{attribute 'linkalways'} 
{attribute 'no_explicit_call' := 'This FB is a CLASS and must be accessed using methods or properties'}
{attribute 'enable_dynamic_creation'}
FUNCTION_BLOCK Node_F_VN_DistanceTransformationExp EXTENDS VisionNode
VAR
    ipSrcImage : _ITcVnImage;
    ipDestImage : _ITcVnImage;
    eDistanceType : _ETcVnDistanceType(ETcVnDistanceType.TCVN_DT_L1);
    eMaskSize : _ETcVnDistanceTransformationMask(ETcVnDistanceTransformationMask.TCVN_DTM_PRECISE);
    ipDestLabels : _ITcVnImage;
    eLabelType : _ETcVnDistanceTransformationLabel(ETcVnDistanceTransformationLabel.TCVN_DTL_CCOMP);
    hrPrev : _HRESULT(S_OK);
	hresult : _HRESULT(S_OK);
END_VAR

METHOD PUBLIC  Clone : I_Node
VAR
	pNode : POINTER TO Node_F_VN_DistanceTransformationExp;
END_VAR
pNode := __NEW(Node_F_VN_DistanceTransformationExp);
Clone := pNode^;
END_METHOD

METHOD FB_init : BOOL
VAR_INPUT
	bInitRetains : BOOL; // if TRUE, the retain variables are initialized (warm start / cold start)
	bInCopyCode : BOOL;  // if TRUE, the instance afterwards gets moved into the copy code (online change)
END_VAR
AddInput('ipSrcImage', ipSrcImage);
AddParameter('eDistanceType', eDistanceType);
AddParameter('eMaskSize', eMaskSize);
AddParameter('eLabelType', eLabelType);
AddInput('hrPrev', hrPrev);
AddOutput('ipDestImage', ipDestImage);
AddOutput('ipDestLabels', ipDestLabels);
AddOutput('hresult',hresult);
END_METHOD

METHOD PROTECTED OnExecute
hresult.Value := F_VN_DistanceTransformationExp(
    ipSrcImage := ipSrcImage.Value,
	ipDestImage := ipDestImage.Value,
    eDistanceType := eDistanceType.Value,
    eMaskSize := eMaskSize.Value,
    ipDestLabels := ipDestLabels.Value,
    eLabelType := eLabelType.Value,
	hrPrev:= hrPrev.Value);
END_METHOD

METHOD PUBLIC PreExecutionCheck
VAR_INPUT
	Check : I_PreExecutionChecks;
END_VAR
VAR
    distanceTypeIsValid : BOOL;
    maskSizeIsValid : BOOL;
END_VAR
Check.IsTrue(ipSrcImage.IsValid, 'ipSrcImage must contain an image');
Check.IsTrue(ipSrcImage.HasChannelCount(1), 'ipSrcImage must have 1 channel');
Check.IsTrue(ipSrcImage.IsPixelDepth(8), 'ipSrcImage must have 8 bit pixel depth');

CASE eDistanceType.Value OF
    ETcVnDistanceType.TCVN_DT_L1,
    ETcVnDistanceType.TCVN_DT_L2,
    ETcVnDistanceType.TCVN_DT_C :
        distanceTypeIsValid := TRUE;
END_CASE
Check.IsTrue(distanceTypeIsValid, 'eDistanceType value is unsupported');

CASE eMaskSize.Value OF
    ETcVnDistanceTransformationMask.TCVN_DTM_3,
    ETcVnDistanceTransformationMask.TCVN_DTM_5 :
        maskSizeIsValid := TRUE;
END_CASE
Check.IsTrue(maskSizeIsValid, 'maskSizeIsValid value is unsupported');
END_METHOD

END_FUNCTION_BLOCK

(* stored: Version 1.1.0.1, ProductVersion 3.1.4024.15
   POU Node_F_VN_DistanceTransformationExp: Id {ff2c9989-7375-4244-a20d-67b814b76b41}, SpecialFunc None
   Folder Constructor: Id {0ac6e05f-fa8b-473e-b8a7-f4d93839d812}
   Method Clone: Id {a38c76e1-8bd5-471a-9be6-96e8afdf7058}
   Method FB_init: Id {8c2b3fa2-0fb1-470f-aa29-b8aedab9ddfb}
   Method OnExecute: Id {4658ab7b-66ba-4928-ad94-a896777df315}
   Method PreExecutionCheck: Id {d486e022-c521-4a60-803c-e4fa6111d44c} *)
